// TIA Portal project "Project13" (V17)

(* hardware
DEVICE "S7-1200 station_1"  S7-1200 Station
   slot 0: "Rack_0"  S7-1200 Rack  Rack  V1.0
   slot 1: "PLC_1"  CPU 1214C DC/DC/DC  6ES7 214-1AG40-0XB0  V4.5
DEVICE "HMI_1"  KTP700 Basic PN
   slot 0: "HMI_1"  KTP700 Basic PN  6AV2 123-2GB03-0AX0  17.0.0.0
   slot 1: "HMI_RT_1"  KTP700 Basic PN  6AV2 123-2GB03-0AX0  17.0.0.0
   slot 5: "HMI_1.IE_CP_1"  PROFINET Interface  17.0.0.0
      slot 1: "PROFINET Interface_1"  PROFINET Interface
         slot 1: "Port_1"  Port
*)

// ===== PLC "PLC_1"  CPU 1214C DC/DC/DC =====

VAR_GLOBAL   // PLC tag table "Default tag table"
   "normalized_temp" AT %M0.0 : LReal;
   "Tag_1" AT %M0.0 : Bool;
END_VAR

VAR_GLOBAL   // PLC tag table "PLC_IO"
   "PB_Start" AT %I0.0 : Bool;   // Momentary Start Button (HMI or Physical)
   "PB_Stop" AT %I0.1 : Bool;   // Momentary Stop Button (HMI or Physical)
   "MainTank_Level_1" AT %I0.2 : Bool;   // Level sensor for Liquid A complete
   "MainTank_Level_2" AT %I0.3 : Bool;   // Level sensor for Liquid B complete (Max Level)
   "MainTank_Level_Low" AT %I0.4 : Bool;   // Low level sensor (Tank empty / Drain complete)
   "Pump1_Overload" AT %I0.5 : Bool;   // Thermal overload relay feedback (Normally Closed)
   "Safety_EStop" AT %I0.6 : Bool;   // Emergency Stop (Normally Closed wiring)
   "Pump1_Run" AT %Q0.0 : Bool;   // Digital command to start Pump 1 contactor
   "MainTank_LiqA_Valve" AT %Q0.1 : Bool;   // Solenoid/Motorized valve for Liquid A
   "MainTank_LiqB_Valve" AT %Q0.2 : Bool;   // Solenoid/Motorized valve for Liquid B
   "MainTank_Heater" AT %Q0.3 : Bool;   // Heating element contactor
   "MainTank_Mixer" AT %Q0.4 : Bool;   // Mixer motor contactor
   "MainTank_Drain_Valve" AT %Q0.5 : Bool;   // Drain valve at the bottom of the tank
   "MainTank_Temp_AI" AT %IW64 : Int;   // Temperature sensor (e.g., 4-20mA scaled to 0-100°C)
END_VAR

DATA_BLOCK "HMI_Commands"   // DB1
{ S7_Optimized_Access := 'FALSE' }
VERSION : 0.1
   VAR
      HMI_Temp_Setpoint : Real := 50.0;
      HMI_Mix_Time_Setpoint : Int := 10000;
      HMI_Start_Cmd : Bool;
      HMI_Stop_Cmd : Bool;
      HMI_Reset_Faults : Bool;
   END_VAR
BEGIN
END_DATA_BLOCK

DATA_BLOCK "Process_Data"   // DB2
{ S7_Optimized_Access := 'FALSE' }
VERSION : 0.1
   VAR
      Current_Step : Int;   // brain of our state machine.
      Actual_Temp : Real := 0.0;
   END_VAR
BEGIN
END_DATA_BLOCK

DATA_BLOCK "Alarm_System"   // DB3
{ S7_Optimized_Access := 'TRUE' }
VERSION : 0.1
   VAR
      Alarm_EStop : Bool;
      Alarm_PumpOverload : Bool;
      Alarm_HighTemp : Bool;
      Alarm_SystemFault : Bool;
      Alarm_Code : Int;
   END_VAR
BEGIN
END_DATA_BLOCK

DATA_BLOCK "FB_Sequence_Controller_DB"   // DB4
{ S7_Optimized_Access := 'TRUE' }
VERSION : 0.1
// stored: InstanceOfName FB_Sequence_Controller
"FB_Sequence_Controller"
BEGIN
END_DATA_BLOCK

DATA_BLOCK "alarm_check_DB"   // DB5
{ S7_Optimized_Access := 'TRUE' }
VERSION : 0.1
// stored: InstanceOfName alarm_check
"alarm_check"
BEGIN
END_DATA_BLOCK

FUNCTION_BLOCK "alarm_check"   // FB1, SCL
{ S7_Optimized_Access := 'TRUE' }
VERSION : 0.1
   VAR_INPUT
      safety_estop : Bool;
      pump_overload : Bool;
   END_VAR
BEGIN

   // --- ALARM CODE GENERATION ---
   // Set individual alarm bits based on conditions

   "Alarm_System".Alarm_EStop := NOT #safety_estop;  // NC contact, so NOT
   "Alarm_System".Alarm_PumpOverload := #pump_overload;
   "Alarm_System".Alarm_HighTemp := ("Process_Data".Actual_Temp > 90.0);
   "Alarm_System".Alarm_SystemFault := ("Process_Data".Current_Step = 99);

   // Calculate combined alarm code (for display on HMI)
   // Each alarm = a specific number
   "Alarm_System".Alarm_Code := 0;

   IF "Alarm_System".Alarm_EStop THEN
       "Alarm_System".Alarm_Code := "Alarm_System".Alarm_Code + 1;
   END_IF;

   IF "Alarm_System".Alarm_PumpOverload THEN
       "Alarm_System".Alarm_Code := "Alarm_System".Alarm_Code + 10;
   END_IF;

   IF "Alarm_System".Alarm_HighTemp THEN
       "Alarm_System".Alarm_Code := "Alarm_System".Alarm_Code + 100;
   END_IF;

   IF "Alarm_System".Alarm_SystemFault THEN
       "Alarm_System".Alarm_Code := "Alarm_System".Alarm_Code + 1000;
   END_IF;
END_FUNCTION_BLOCK

FUNCTION_BLOCK "FB_Sequence_Controller"   // FB2, SCL
{ S7_Optimized_Access := 'TRUE' }
VERSION : 0.1
   VAR_INPUT
      pump_overload : Bool;
      MainTank_Level_1 : Bool;
      MainTank_Level_2 : Bool;
      MainTank_Level_low : Bool;
   END_VAR
   VAR_OUTPUT
      pump1_run : Bool;
      MainTank_LiqA_valve : Bool;
      MainTank_LiqB_valve : Bool;
      MainTank_heater : Bool;
      MainTank_mixer : Bool;
      MainTank_drain_valve : Bool;
   END_VAR
   VAR_IN_OUT
      temp_hmi_setpoint : Real;
      actual_temp : Real;
      current_step : Int;
      reset_fault : Bool;
      start_btn : Bool;
      safety_Estop : Bool;
      stop_btn : Bool;
      mix_time_setpoint : Int;
   END_VAR
   VAR
      mix_timer : IEC_TIMER;
   END_VAR
   VAR_TEMP
      time_set_point_time : Time;
   END_VAR
BEGIN
   IF #safety_Estop OR #pump_overload OR #stop_btn THEN
       #current_step := 99
       ;
   END_IF;
   // --- 2. STATE MACHINE ---
   CASE #current_step OF
       0:  // IDLE (Waiting for Start)
           // Turn off all outputs to ensure safe state
           #pump1_run := FALSE;
           #MainTank_LiqA_valve := FALSE;
           #MainTank_LiqB_valve := FALSE;
           #MainTank_heater := FALSE;
           #MainTank_mixer := FALSE;
           #MainTank_drain_valve := FALSE;
           IF #start_btn THEN
               #current_step := 10;
           END_IF;

       10:  // Fill liquid A
           #pump1_run := TRUE;
           #MainTank_LiqA_valve := TRUE;
           IF #MainTank_Level_1 THEN
               #pump1_run := FALSE;
               #MainTank_LiqA_valve := FALSE;
               #current_step := 20;
           END_IF;
       20: // Fill liquid B
           #MainTank_LiqB_valve := TRUE;
           IF #MainTank_Level_2 THEN
               #MainTank_LiqB_valve := FALSE;
               #current_step := 30;
           END_IF;
       30: // Heating
           #MainTank_heater := TRUE;
           IF #actual_temp >= #temp_hmi_setpoint THEN
               #MainTank_heater := FALSE;
               #current_step := 40;
               ;
           END_IF;


           ;
       40: // MIXER
           #MainTank_mixer := TRUE;

           #time_set_point_time:= INT_TO_TIME(#mix_time_setpoint);

           #mix_timer.TON(IN:= TRUE,
                          PT:= #time_set_point_time );
           IF #mix_timer.Q THEN
               #mix_timer.TON(IN := FALSE, PT:= #time_set_point_time);
               #MainTank_mixer := FALSE;
               #current_step := 50;
               ;
           END_IF;

       50: // DRAINING
           #MainTank_drain_valve := TRUE;
           IF #MainTank_Level_low THEN
               #MainTank_drain_valve := FALSE;
               #current_step := 0;
               ;
           END_IF;
       99: // ERROR
           #pump1_run := FALSE;
           #MainTank_LiqA_valve := FALSE;
           #MainTank_LiqB_valve := FALSE;
           #MainTank_heater := FALSE;
           #MainTank_mixer := FALSE;
           #MainTank_drain_valve := FALSE;
           IF #reset_fault THEN
               #current_step := 0;
           END_IF;
           ;
   END_CASE;
END_FUNCTION_BLOCK

ORGANIZATION_BLOCK "Main"   // OB1, LAD, ProgramCycle
TITLE = "Main Program Sweep (Cycle)"
{ S7_Optimized_Access := 'TRUE' }
VERSION : 0.1
   VAR_INPUT
      Initial_Call : Bool;   // Initial call of this OB
      Remanence : Bool;   // =True, if remanent data are available
   END_VAR
BEGIN

REGION Network 1
   // temperature Analog Scaling
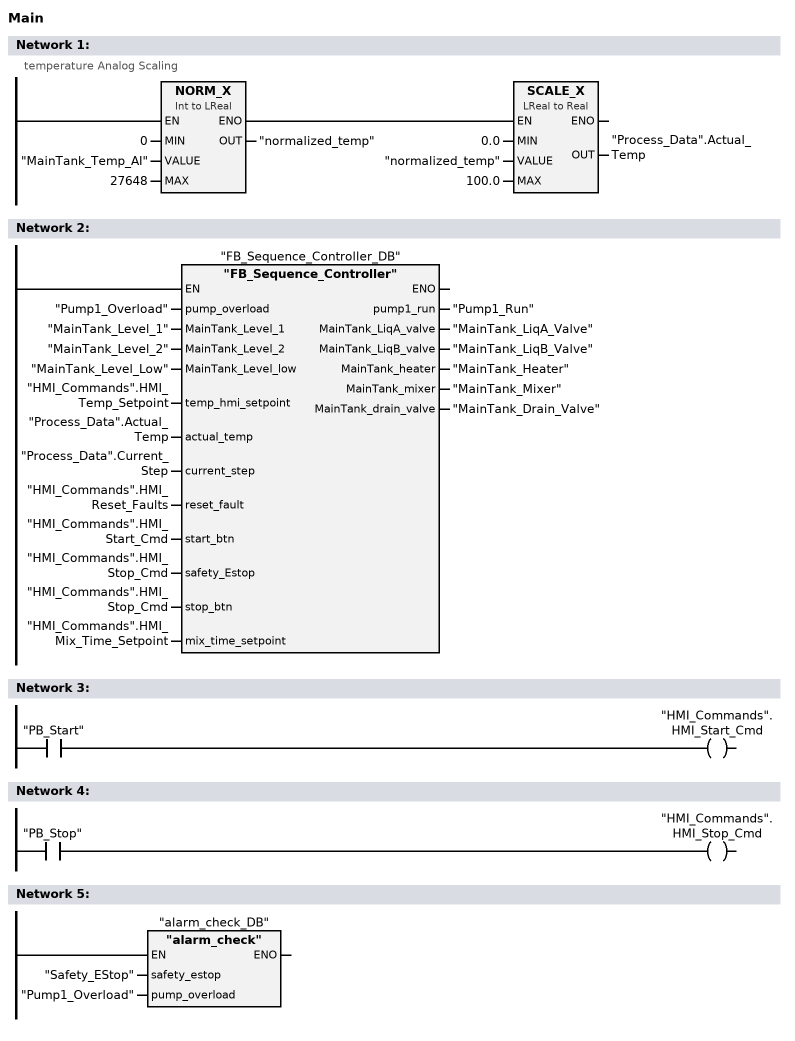
   RUNG wire#powerrail
      { S7_Templates := "[SrcType := Int, DestType := LReal]" } Normalize(min := 0, value := "MainTank_Temp_AI", max := 27648, out => "normalized_temp")
      { S7_Templates := "[SrcType := LReal, DestType := Real]" } Scale(min := 0.0, value := "normalized_temp", max := 100.0, out => "Process_Data".Actual_Temp)
   END_RUNG
   // the same network as SCL:
   "normalized_temp" := NORM_X(MIN := 0, VALUE := "MainTank_Temp_AI", MAX := 27648);
   "Process_Data".Actual_Temp := SCALE_X(MIN := 0.0, VALUE := "normalized_temp", MAX := 100.0);
END_REGION

REGION Network 2
   RUNG wire#powerrail
      "FB_Sequence_Controller_DB"(pump_overload := "Pump1_Overload", MainTank_Level_1 := "MainTank_Level_1", MainTank_Level_2 := "MainTank_Level_2", MainTank_Level_low := "MainTank_Level_Low", temp_hmi_setpoint := "HMI_Commands".HMI_Temp_Setpoint, actual_temp := "Process_Data".Actual_Temp, current_step := "Process_Data".Current_Step, reset_fault := "HMI_Commands".HMI_Reset_Faults, start_btn := "HMI_Commands".HMI_Start_Cmd, safety_Estop := "HMI_Commands".HMI_Stop_Cmd, stop_btn := "HMI_Commands".HMI_Stop_Cmd, mix_time_setpoint := "HMI_Commands".HMI_Mix_Time_Setpoint, pump1_run => "Pump1_Run", MainTank_LiqA_valve => "MainTank_LiqA_Valve", MainTank_LiqB_valve => "MainTank_LiqB_Valve", MainTank_heater => "MainTank_Heater", MainTank_mixer => "MainTank_Mixer", MainTank_drain_valve => "MainTank_Drain_Valve")
   END_RUNG
   // the same network as SCL:
   "FB_Sequence_Controller_DB"(pump_overload := "Pump1_Overload",   // "FB_Sequence_Controller"
                           MainTank_Level_1 := "MainTank_Level_1",
                           MainTank_Level_2 := "MainTank_Level_2",
                           MainTank_Level_low := "MainTank_Level_Low",
                           temp_hmi_setpoint := "HMI_Commands".HMI_Temp_Setpoint,
                           actual_temp := "Process_Data".Actual_Temp,
                           current_step := "Process_Data".Current_Step,
                           reset_fault := "HMI_Commands".HMI_Reset_Faults,
                           start_btn := "HMI_Commands".HMI_Start_Cmd,
                           safety_Estop := "HMI_Commands".HMI_Stop_Cmd,
                           stop_btn := "HMI_Commands".HMI_Stop_Cmd,
                           mix_time_setpoint := "HMI_Commands".HMI_Mix_Time_Setpoint,
                           pump1_run => "Pump1_Run",
                           MainTank_LiqA_valve => "MainTank_LiqA_Valve",
                           MainTank_LiqB_valve => "MainTank_LiqB_Valve",
                           MainTank_heater => "MainTank_Heater",
                           MainTank_mixer => "MainTank_Mixer",
                           MainTank_drain_valve => "MainTank_Drain_Valve");
END_REGION

REGION Network 3
   RUNG wire#powerrail
      Contact( "PB_Start" )
      Coil( "HMI_Commands".HMI_Start_Cmd )
   END_RUNG
   // the same network as SCL:
   "HMI_Commands".HMI_Start_Cmd := "PB_Start";
END_REGION

REGION Network 4
   RUNG wire#powerrail
      Contact( "PB_Stop" )
      Coil( "HMI_Commands".HMI_Stop_Cmd )
   END_RUNG
   // the same network as SCL:
   "HMI_Commands".HMI_Stop_Cmd := "PB_Stop";
END_REGION

REGION Network 5
   RUNG wire#powerrail
      "alarm_check_DB"(safety_estop := "Safety_EStop", pump_overload := "Pump1_Overload")
   END_RUNG
   // the same network as SCL:
   "alarm_check_DB"(safety_estop := "Safety_EStop", pump_overload := "Pump1_Overload");   // "alarm_check"
END_REGION
END_ORGANIZATION_BLOCK

(* ===== HMI "HMI_RT_1" =====
system functions are stored by id; their names below are inferred from use
connection "HMI_Connection_1": ETHERNET, SMART_S7_1200_OMS

HMI tags "Default tag table"
   "Safety_EStop" : Bool = PLC Safety_EStop AT %I0.6, 1 s
   "FB_Sequence_Controller_DB_mix_timer_PT" : Time = PLC FB_Sequence_Controller_DB.mix_timer.PT, 1 s

HMI tags "PLC_Connection"
   "HMI_Commands_HMI_Start_Cmd" : Bool = PLC HMI_Commands.HMI_Start_Cmd AT %DB1.DBX6.0, 1 s
   "HMI_Commands_HMI_Stop_Cmd" : Bool = PLC HMI_Commands.HMI_Stop_Cmd AT %DB1.DBX6.1, 1 s
   "HMI_Commands_HMI_Reset_Faults" : Bool = PLC HMI_Commands.HMI_Reset_Faults AT %DB1.DBX6.2, 1 s
   "HMI_Commands_HMI_Mix_Time_Setpoint" : Int = PLC HMI_Commands.HMI_Mix_Time_Setpoint AT %DB1.DBW4, 1 s
   "HMI_Commands_HMI_Temp_Setpoint" : Real = PLC HMI_Commands.HMI_Temp_Setpoint AT %DB1.DBD0, 1 s
   "Process_Data_Current_Step" : Int = PLC Process_Data.Current_Step AT %DB2.DBW0, 1 s
   "Process_Data_Actual_Temp" : Real = PLC Process_Data.Actual_Temp AT %DB2.DBD2, 1 s
   "Pump1_Run" : Bool = PLC Pump1_Run AT %Q0.0, 1 s
   "MainTank_LiqA_Valve" : Bool = PLC MainTank_LiqA_Valve AT %Q0.1, 1 s
   "MainTank_LiqB_Valve" : Bool = PLC MainTank_LiqB_Valve AT %Q0.2, 1 s
   "MainTank_Mixer" : Bool = PLC MainTank_Mixer AT %Q0.4, 1 s
   "MainTank_Heater" : Bool = PLC MainTank_Heater AT %Q0.3, 1 s
   "MainTank_Drain_Valve" : Bool = PLC MainTank_Drain_Valve AT %Q0.5, 1 s
   "MainTank_Level_1" : Bool = PLC MainTank_Level_1 AT %I0.2, 1 s
   "MainTank_Level_2" : Bool = PLC MainTank_Level_2 AT %I0.3, 1 s
   "MainTank_Level_Low" : Bool = PLC MainTank_Level_Low AT %I0.4, 1 s

HMI tags "Tag table_1"
   "Alarm_System_Alarm_Code" : Int = PLC Alarm_System.Alarm_Code, 1 s

discrete alarms
   1: 'ALARM 001: EMERGENCY STOP ACTIVATED / The sensor is broken', class Errors, trigger "Alarm_System_Alarm_Code" bit 0
   4: 'ALARM 004: SYSTEM FAULT - Check step 99', class Errors, trigger "Alarm_System_Alarm_Code" bit 3
   2: 'ALARM 002: PUMP MOTOR OVERLOAD', class Errors, trigger "Alarm_System_Alarm_Code" bit 1
   3: 'ALARM 003: HIGH TEMPERATURE WARNING', class Errors, trigger "Alarm_System_Alarm_Code" bit 2

analog alarms
   1: 'HIGH TEMPERATURE REACHED', class Warnings, trigger "Process_Data_Actual_Temp"

screen "Main_Overview" 800x480
   TextField "Text field_1" at 252,2 size 320x34; Text 'Liquid Batching System'
   TextField "Text field_2" at 35,79 size 104x23; Text 'Current step'
   IOField "I/O field_1" at 157,73 size 96x32; FormatPattern 99
      ProcessValue <- "Process_Data_Current_Step"
   TextField "Text field_3" at 348,61 size 50x23; Text 'Pump'
   TextField "Text field_4" at 264,124 size 76x23; Text 'VALVE A'
   TextField "Text field_5" at 419,125 size 74x23; Text 'VALVE B'
   Line "Line_1" at 326,155 size 0x39
      Visibility <- "MainTank_LiqA_Valve"
   Line "Line_2" at 431,157 size 0x39
      Visibility <- "MainTank_LiqB_Valve"
   Line "Line_3" at 360,371 size 59x1
      Visibility <- "MainTank_Drain_Valve"
   TextField "Text field_6" at 347,399 size 118x23; Text 'DRAIN VALVE'
   Line "Line_4" at 375,220 size 1x98
      Appearance <- "MainTank_Mixer"
   Ellipse "Ellipse_2" at 343,311 size 72x24
      Appearance <- "MainTank_Mixer"
   TextField "Text field_7" at 348,194 size 56x23; Text 'MIXER'
   TextField "Text field_8" at 455,279 size 71x23; Text 'HEATER'
   Button "Button_1" at 4,439 size 96x32; TextOff 'START'
      on Press: SetBit("HMI_Commands_HMI_Start_Cmd")
      on Release: ResetBit("HMI_Commands_HMI_Start_Cmd")
   Button "Button_2" at 110,438 size 96x32; TextOff 'STOP'
      on Release: ResetBit("HMI_Commands_HMI_Stop_Cmd")
      on Press: SetBit("HMI_Commands_HMI_Stop_Cmd")
   Button "Button_3" at 226,438 size 96x32; TextOff 'RESET'
      on Release: ResetBit("HMI_Commands_HMI_Reset_Faults")
      on Press: SetBit("HMI_Commands_HMI_Reset_Faults")
   IOField "I/O field_2" at 663,61 size 96x32; FormatPattern 99999
      ProcessValue <- "HMI_Commands_HMI_Temp_Setpoint"
   TextField "Text field_9" at 611,35 size 163x23; Text 'TEMP SETPOINT'
   TextField "Text field_10" at 607,103 size 186x23; Text 'Mix Time Setpoint'
   IOField "I/O field_3" at 663,134 size 96x32; FormatPattern 99999
      ProcessValue <- "HMI_Commands_HMI_Mix_Time_Setpoint"
   TextField "Text field_11" at 623,182 size 106x23; Text 'Actual Temp'
   IOField "I/O field_4" at 663,213 size 96x32; FormatPattern s999999999.999
      ProcessValue <- "Process_Data_Actual_Temp"
   TextField "Text field_12" at 759,209 size 25x23; Text '°C'
   Ellipse "Ellipse_3" at 341,79 size 78x53
      Appearance <- "Pump1_Run"
   Ellipse "Ellipse_4" at 443,303 size 75x32
      Appearance <- "MainTank_Heater"
   Line "Line_5" at 231,280 size 57x0
      Appearance <- "MainTank_Level_1"
   TextField "Text field_13" at 231,359 size 95x23; Text 'sensor Low'
   TextField "Text field_14" at 477,224 size 73x23; Text 'sensor B'
   Line "Line_6" at 461,223 size 57x0
      Appearance <- "MainTank_Level_2"
   Line "Line_7" at 265,352 size 57x0
      Appearance <- "MainTank_Level_Low"
   TextField "Text field_15" at 206,288 size 75x23; Text 'sensor A'
   Button "Button_4" at 697,439 size 96x32; TextOff 'ALARMS'
      on Click: ActivateScreen("Alarms", 0)
   Button "Button_5" at 578,440 size 96x32; TextOff 'TRENDS'
      on Click: ActivateScreen("Trends", 0)

screen "Alarms" 800x480
   AlarmView "Alarm view_1" at 63,45 size 649x315
   Button "Button_1" at 67,435 size 96x32; TextOff 'Home'
      on Click: ActivateScreen("Main_Overview", 0)
   Button "Button_5" at 178,435 size 96x32; TextOff 'TRENDS'
      on Click: ActivateScreen("Trends", 0)

screen "Trends" 800x480
   TrendView "Trend view_1" at 59,16 size 688x372
   Button "Button_4" at 27,417 size 96x32; TextOff 'ALARMS'
      on Click: ActivateScreen("Alarms", 0)
   Button "Button_1" at 152,417 size 96x32; TextOff 'Home'
      on Click: ActivateScreen("Main_Overview", 0)
*)